// Mitsubishi GX Works2 project: NOR   PLC: Q03UDV

PROGRAM MAIN
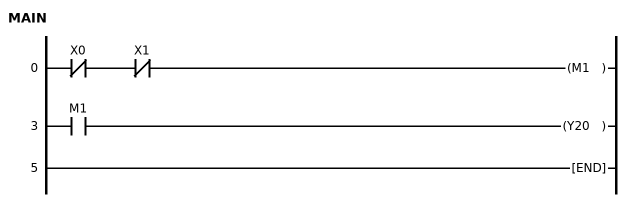
0     LDI     X0
      ANI     X1
      OUT     M1
3     LD      M1
      OUT     Y20
5     END
END_PROGRAM
